(*
SPDX-FileCopyrightText: © 2026 Oleksandr Tiutyk <trofimich@gmail.com>
SPDX-License-Identifier: MIT
License: https://opensource.org/license/mit
*)

INTERFACE ITargetVariableMemoryOverflowException EXTENDS IGeneralException

METHOD Throw
VAR_INPUT
	sourceNamespaceName : STRING;
	sourceClassName : STRING;
	sourcePOUName : STRING;
	sourcePosition : STRING;
	targetVariableName : STRING;
	targetVariableSize : ULINT;
END_VAR
END_METHOD

END_INTERFACE

(* stored: Version 1.1.0.1
   Itf ITargetVariableMemoryOverflowException: Id {39f9ecfc-89ca-4ccd-9c46-c14c94c08b7f}
   Method Throw: Id {c2c590e2-59c3-4764-8971-347504c00428} *)
